// TIA Portal V18 export
// export: Created 2026-06-16T05:09:48.1075673Z, ExportSetting WithDefaults, DisplayName Totally Integrated Automation Portal, DisplayVersion V18 Update 5, DisplayName TIA Portal Openness, DisplayVersion V18 Update 5, DisplayName TIA Portal Version Control Interface, DisplayVersion V18, DisplayName SINAMICS Startdrive Advanced, DisplayVersion V18 SP2 Update 1, DisplayName SINAMICS Startdrive G110M, G120, G120C, G120D, G120P, G115D, DisplayVersion V18 SP2 Update 1, DisplayName SINAMICS Startdrive G130, G150, S120, S150, SINAMICS MV, S210, G220, S200, DisplayVersion V18 SP2 Update 1, DisplayName STEP 7 Professional, DisplayVersion V18 Update 5, DisplayName STEP 7 Safety, DisplayVersion V18, DisplayName WinCC Advanced / Unified PC, DisplayVersion V18 Update 5
FUNCTION "TEMPLATE--v1.1--00_Only for Commissioning" : Void   // FC4, F_LAD
TITLE = bypass activation by profinet node to use during commissioning
{ S7_Optimized_Access := 'TRUE' }
VERSION : 0.1
// 1.0 First Emission
// 1.1 Aligned Syntax to signal_types.csv of the py_builder
// stored: AutoNumber true, IsIECCheckEnabled false, UDAEnableTagReadback false
BEGIN

REGION Network 1: !!NetworkComment$$
   // One network per node
   // TRUE if the node is not ready to be used
   // FALSE if the node is ready
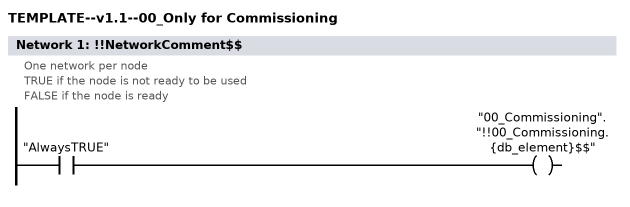
   RUNG wire#powerrail
      Contact( "AlwaysTRUE" )
      Coil( "00_Commissioning"."!!00_Commissioning.{db_element}$$" )
   END_RUNG
   // the same network as SCL:
   "00_Commissioning"."!!00_Commissioning.{db_element}$$" := "AlwaysTRUE";
END_REGION
END_FUNCTION
